SUBAPPLICATION Uebung_012l (* String Input und Speichern NVS *)
  (* Standard: 61499-2; Description: Copyright (c) 2023 Meisterschulen am Ostbahnhof This program and the accompanying materials are made available under the terms of the Eclipse Public License 2.0 which is available at https://www.eclipse.org/legal/epl-2.0/ SPDX-License-Identifier: EPL-2.0 *)
  (* Version 1.0, 2023-10-23, Franz Höpfinger, Meisterschulen am Ostbahnhof, initial API and implementation and/or initial documentation *)
  PACKAGE Uebungen;
  IMPORT Uebungen::const::NVS::NVS_Keys::KEY_S1_STORE;
  IMPORT Uebungen::const::UT::DefaultPool::InputString_S1;
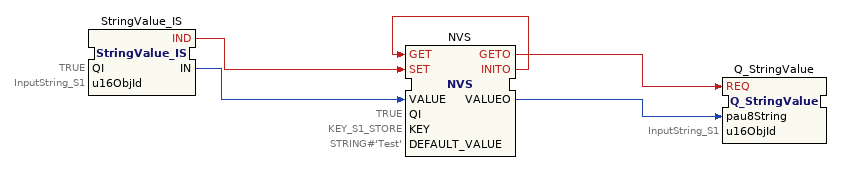
  FBS
    StringValue_IS : isobus::UT::io::StringValue::StringValue_IS(QI := TRUE, u16ObjId := InputString_S1);
    NVS : logiBUS::storage::esp32_nvs::NVS(QI := TRUE, KEY := KEY_S1_STORE, DEFAULT_VALUE := STRING#'Test');
    Q_StringValue : isobus::UT::Q::Q_StringValue(u16ObjId := InputString_S1);
  END_FBS
  EVENT_CONNECTIONS
    NVS.GETO TO Q_StringValue.REQ;
    NVS.INITO TO NVS.GET;
    StringValue_IS.IND TO NVS.SET;
  END_CONNECTIONS
  DATA_CONNECTIONS
    NVS.VALUEO TO Q_StringValue.pau8String;
    StringValue_IS.IN TO NVS.VALUE;
  END_CONNECTIONS
END_SUBAPPLICATION
